// TIA Portal project "Hệ thống bơm cấp nước" (V16)

(* hardware
DEVICE "PC-System_1"  SIMATIC PC station
   slot 0: "SIMATIC PC station"  Rail  SIMATIC PC-Station  V1.0
      slot 125: "Stationmanager"  Station_Manager  V6.0.4
   slot 1: "HMI_RT_1"  WinCC RT Advanced  6AV2 104-0xxxx-xxxx  16.0.0.0
      slot 33792: "Computer interface"  Host interface
   slot 2: "IE general_1"  IE General  IE_CP  V8.2.0
DEVICE "S7-1200 station_1"  S7-1200 Station
   slot 0: "Rack_0"  S7-1200 Rack  Rack  V1.0
   slot 1: "PLC_1"  CPU 1214C DC/DC/DC  6ES7 214-1AG40-0XB0  V4.4
DEVICE "PC-System_2"  SIMATIC PC station
   slot 0: "SIMATIC PC station"  Rail  SIMATIC PC-Station  V1.0
      slot 125: "Stationmanager"  Station_Manager  V6.0.4
   slot 2: "IE general_1"  IE General  IE_CP  V8.2.0
*)

// ===== PLC "PLC_1"  CPU 1214C DC/DC/DC =====

VAR_GLOBAL   // PLC tag table "Default tag table"
   "START_VALVE_1" AT %M3.0 : Bool;
   "STOP_VALVE_1" AT %M3.1 : Bool;
   "START_VALVE_2" AT %M3.2 : Bool;
   "STOP_VALVE_2" AT %M3.3 : Bool;
   "START_PUMP_1" AT %M3.4 : Bool;
   "STOP_PUMP_1" AT %M3.5 : Bool;
   "START_PUMP_2" AT %M3.6 : Bool;
   "STOP_PUMP_2" AT %M3.7 : Bool;
   "START_PUMP_SUPPLY" AT %M4.0 : Bool;
   "STOP_PUMP_SUPPLY" AT %M4.1 : Bool;
   "VALVE_1" AT %Q0.0 : Bool;
   "VALVE_2" AT %Q0.1 : Bool;
   "PUMP_1" AT %Q0.2 : Bool;
   "PUMP_2" AT %Q0.3 : Bool;
   "PUMP_SUPPLY" AT %Q0.4 : Bool;
   "VALUE" AT %M4.2 : Bool;
   "SENSOR_1" AT %M4.3 : Bool;
   "SENSOR_2" AT %M4.4 : Bool;
   "SENSOR_3" AT %M4.5 : Bool;
   "TIME_RUN_PUMP 1" AT %MD10 : Time;
   "NO_WATER_PUMP_1" AT %M4.6 : Bool;
   "NO_WATER_PUMP_2" AT %M4.7 : Bool;
   "TIME_RUN_PUMP 2" AT %MD14 : Time;
   "System_Byte" AT %MB1 : Byte;
   "FirstScan" AT %M1.0 : Bool;
   "DiagStatusUpdate" AT %M1.1 : Bool;
   "AlwaysTRUE" AT %M1.2 : Bool;
   "AlwaysFALSE" AT %M1.3 : Bool;
   "Clock_Byte" AT %MB0 : Byte;
   "Clock_10Hz" AT %M0.0 : Bool;
   "Clock_5Hz" AT %M0.1 : Bool;
   "Clock_2.5Hz" AT %M0.2 : Bool;
   "Clock_2Hz" AT %M0.3 : Bool;
   "Clock_1.25Hz" AT %M0.4 : Bool;
   "Clock_1Hz" AT %M0.5 : Bool;
   "Clock_0.625Hz" AT %M0.6 : Bool;
   "Clock_0.5Hz" AT %M0.7 : Bool;
   "FULL_TANK_TOP" AT %M5.0 : Bool;
   "LEVEL_TANK_TOP" AT %MW18 : UInt;
   "EMPTY_TANK_TOP" AT %M5.1 : Bool;
   "FULL_TANK_BOT" AT %M5.2 : Bool;
   "USER" AT %MW22 : Word;
   "LEVEL_TANK_BOT" AT %MW20 : UInt;
   "EMPTY_TANK_BOT" AT %M5.3 : Bool;
END_VAR

// folder: System blocks/Program resources

DATA_BLOCK "IEC_Timer_0_DB"   // DB1
{ S7_Optimized_Access := 'TRUE' }
AUTHOR : Simatic
FAMILY : IEC
NAME : IEC_TMR
VERSION : 1.0
// stored: InstanceOfName IEC_TIMER
"IEC_TIMER"
BEGIN
END_DATA_BLOCK

DATA_BLOCK "IEC_Timer_0_DB_1"   // DB2
{ S7_Optimized_Access := 'TRUE' }
AUTHOR : Simatic
FAMILY : IEC
NAME : IEC_TMR
VERSION : 1.0
// stored: InstanceOfName IEC_TIMER
"IEC_TIMER"
BEGIN
END_DATA_BLOCK

DATA_BLOCK "IEC_Counter_0_DB"   // DB3
{ S7_Optimized_Access := 'TRUE' }
AUTHOR : Simatic
FAMILY : IEC
NAME : UCNTR
VERSION : 1.2
// stored: InstanceOfName IEC_UCOUNTER
"IEC_UCOUNTER"
BEGIN
END_DATA_BLOCK

DATA_BLOCK "IEC_Counter_0_DB_1"   // DB4
{ S7_Optimized_Access := 'TRUE' }
AUTHOR : Simatic
FAMILY : IEC
NAME : UCNTR
VERSION : 1.2
// stored: InstanceOfName IEC_UCOUNTER
"IEC_UCOUNTER"
BEGIN
END_DATA_BLOCK

// folder: (top level)

ORGANIZATION_BLOCK "Main"   // OB1, LAD, ProgramCycle
TITLE = Hệ thống cung cấp nước
{ S7_Optimized_Access := 'TRUE' }
VERSION : 0.1
   VAR_INPUT
      Initial_Call : Bool;   // Initial call of this OB
      Remanence : Bool;   // =True, if remanent data are available
   END_VAR
   VAR_TEMP
      EMPTY_TANK_BOT : Bool;
      LEVEL_TANK_BOT : Int;
   END_VAR
BEGIN

REGION Network 1: Control valve 1
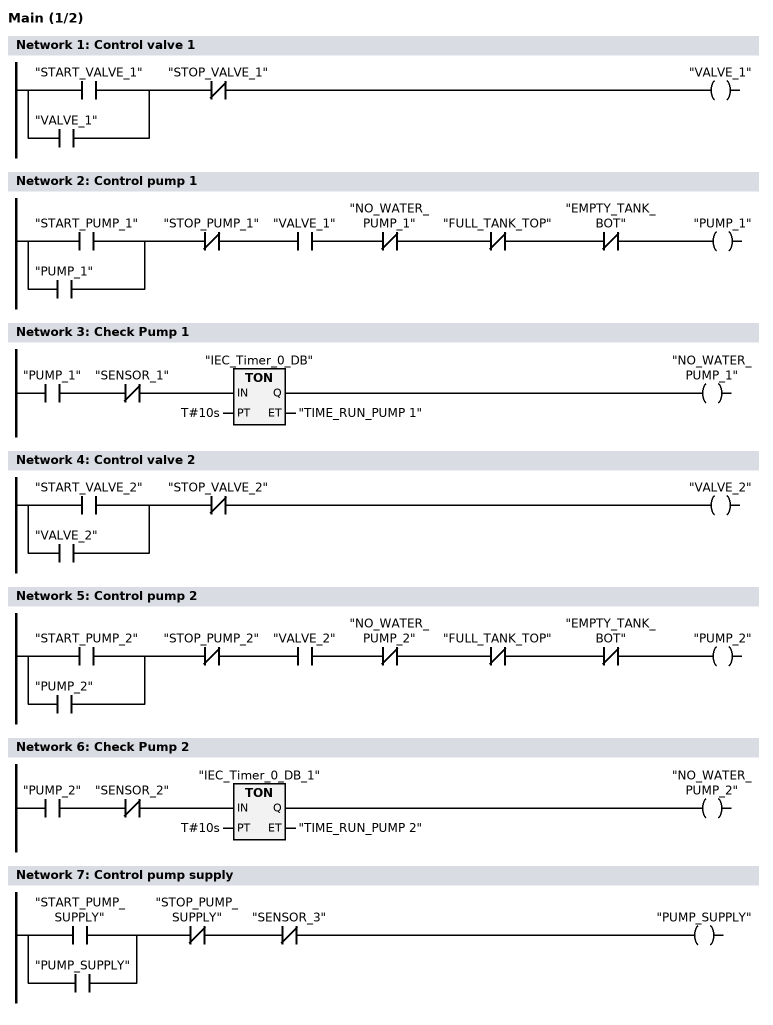
   RUNG wire#powerrail
      Contact( "START_VALVE_1" )
      wire#w1
      I_Contact( "STOP_VALVE_1" )
      Coil( "VALVE_1" )
   END_RUNG
   RUNG wire#powerrail
      Contact( "VALVE_1" )
   END_RUNG wire#w1
   // the same network as SCL:
   "VALVE_1" := ("START_VALVE_1" OR "VALVE_1") AND NOT "STOP_VALVE_1";
END_REGION

REGION Network 2: Control pump 1
   RUNG wire#powerrail
      Contact( "START_PUMP_1" )
      wire#w1
      I_Contact( "STOP_PUMP_1" )
      Contact( "VALVE_1" )
      I_Contact( "NO_WATER_PUMP_1" )
      I_Contact( "FULL_TANK_TOP" )
      I_Contact( "EMPTY_TANK_BOT" )
      Coil( "PUMP_1" )
   END_RUNG
   RUNG wire#powerrail
      Contact( "PUMP_1" )
   END_RUNG wire#w1
   // the same network as SCL:
   "PUMP_1" := ("START_PUMP_1" OR "PUMP_1") AND NOT "STOP_PUMP_1" AND "VALVE_1" AND NOT "NO_WATER_PUMP_1" AND NOT "FULL_TANK_TOP" AND NOT "EMPTY_TANK_BOT";
END_REGION

REGION Network 3: Check Pump 1
   "IEC_Timer_0_DB".TON(IN := "PUMP_1" AND NOT "SENSOR_1", PT := T#10s, ET => "TIME_RUN_PUMP 1");
   "NO_WATER_PUMP_1" := "IEC_Timer_0_DB".Q;
END_REGION

REGION Network 4: Control valve 2
   RUNG wire#powerrail
      Contact( "START_VALVE_2" )
      wire#w1
      I_Contact( "STOP_VALVE_2" )
      Coil( "VALVE_2" )
   END_RUNG
   RUNG wire#powerrail
      Contact( "VALVE_2" )
   END_RUNG wire#w1
   // the same network as SCL:
   "VALVE_2" := ("START_VALVE_2" OR "VALVE_2") AND NOT "STOP_VALVE_2";
END_REGION

REGION Network 5: Control pump 2
   RUNG wire#powerrail
      Contact( "START_PUMP_2" )
      wire#w1
      I_Contact( "STOP_PUMP_2" )
      Contact( "VALVE_2" )
      I_Contact( "NO_WATER_PUMP_2" )
      I_Contact( "FULL_TANK_TOP" )
      I_Contact( "EMPTY_TANK_BOT" )
      Coil( "PUMP_2" )
   END_RUNG
   RUNG wire#powerrail
      Contact( "PUMP_2" )
   END_RUNG wire#w1
   // the same network as SCL:
   "PUMP_2" := ("START_PUMP_2" OR "PUMP_2") AND NOT "STOP_PUMP_2" AND "VALVE_2" AND NOT "NO_WATER_PUMP_2" AND NOT "FULL_TANK_TOP" AND NOT "EMPTY_TANK_BOT";
END_REGION

REGION Network 6: Check Pump 2
   "IEC_Timer_0_DB_1".TON(IN := "PUMP_2" AND NOT "SENSOR_2", PT := T#10s, ET => "TIME_RUN_PUMP 2");
   "NO_WATER_PUMP_2" := "IEC_Timer_0_DB_1".Q;
END_REGION

REGION Network 7: Control pump supply
   RUNG wire#powerrail
      Contact( "START_PUMP_SUPPLY" )
      wire#w1
      I_Contact( "STOP_PUMP_SUPPLY" )
      I_Contact( "SENSOR_3" )
      Coil( "PUMP_SUPPLY" )
   END_RUNG
   RUNG wire#powerrail
      Contact( "PUMP_SUPPLY" )
   END_RUNG wire#w1
   // the same network as SCL:
   "PUMP_SUPPLY" := ("START_PUMP_SUPPLY" OR "PUMP_SUPPLY") AND NOT "STOP_PUMP_SUPPLY" AND NOT "SENSOR_3";
END_REGION

REGION Network 8: Simulation tank top
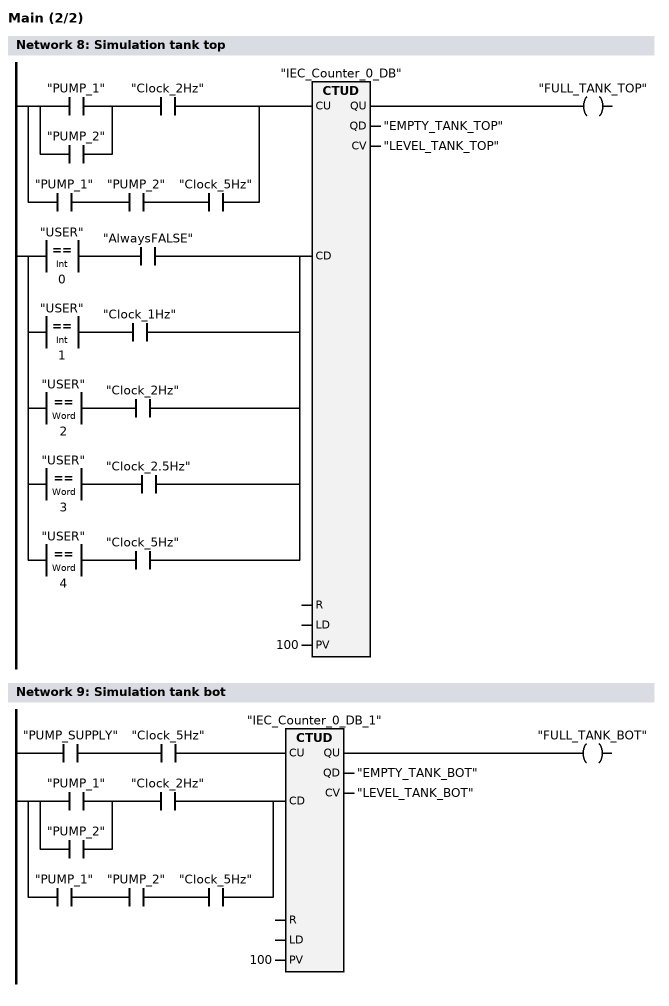
   "IEC_Counter_0_DB".CTUD(CU := (("PUMP_1" OR "PUMP_2") AND "Clock_2Hz") OR ("PUMP_1" AND "PUMP_2" AND "Clock_5Hz"),
                           CD := (("USER" = 0) AND "AlwaysFALSE") OR (("USER" = 1) AND "Clock_1Hz") OR (("USER" = 2) AND "Clock_2Hz") OR (("USER" = 3) AND "Clock_2.5Hz") OR (("USER" = 4) AND "Clock_5Hz"),
                           PV := 100,
                           QD => "EMPTY_TANK_TOP",
                           CV => "LEVEL_TANK_TOP");
   "FULL_TANK_TOP" := "IEC_Counter_0_DB".QU;
END_REGION

REGION Network 9: Simulation tank bot
   "IEC_Counter_0_DB_1".CTUD(CU := "PUMP_SUPPLY" AND "Clock_5Hz",
                           CD := (("PUMP_1" OR "PUMP_2") AND "Clock_2Hz") OR ("PUMP_1" AND "PUMP_2" AND "Clock_5Hz"),
                           PV := 100,
                           QD => "EMPTY_TANK_BOT",
                           CV => "LEVEL_TANK_BOT");
   "FULL_TANK_BOT" := "IEC_Counter_0_DB_1".QU;
END_REGION
END_ORGANIZATION_BLOCK

(* ===== HMI "HMI_RT_1" =====
system functions are stored by id; their names below are inferred from use
connection "HMI_Connection_1": ETHERNET, S7_1200_OMS

HMI tags "Default tag table"
   "START_VALVE_1" : Bool = PLC START_VALVE_1 AT %M3.0, 1 s
   "STOP_VALVE_1" : Bool = PLC STOP_VALVE_1 AT %M3.1, 1 s
   "START_VALVE_2" : Bool = PLC START_VALVE_2 AT %M3.2, 1 s
   "STOP_VALVE_2" : Bool = PLC STOP_VALVE_2 AT %M3.3, 1 s
   "START_PUMP_1" : Bool = PLC START_PUMP_1 AT %M3.4, 1 s
   "STOP_PUMP_1" : Bool = PLC STOP_PUMP_1 AT %M3.5, 1 s
   "START_PUMP_2" : Bool = PLC START_PUMP_2 AT %M3.6, 1 s
   "STOP_PUMP_2" : Bool = PLC STOP_PUMP_2 AT %M3.7, 1 s
   "START_PUMP_SUPPLY" : Bool = PLC START_PUMP_SUPPLY AT %M4.0, 1 s
   "STOP_PUMP_SUPPLY" : Bool = PLC STOP_PUMP_SUPPLY AT %M4.1, 1 s
   "VALVE_1" : Bool = PLC VALVE_1 AT %Q0.0, 1 s
   "VALVE_2" : Bool = PLC VALVE_2 AT %Q0.1, 1 s
   "PUMP_1" : Bool = PLC PUMP_1 AT %Q0.2, 1 s
   "PUMP_2" : Bool = PLC PUMP_2 AT %Q0.3, 1 s
   "PUMP_SUPPLY" : Bool = PLC PUMP_SUPPLY AT %Q0.4, 1 s
   "VALUE" : Bool = PLC VALUE AT %M4.2, 1 s
   "SENSOR_1" : Bool = PLC SENSOR_1 AT %M4.3, 1 s
   "SENSOR_2" : Bool = PLC SENSOR_2 AT %M4.4, 1 s
   "SENSOR_3" : Bool = PLC SENSOR_3 AT %M4.5, 1 s
   "TIME_RUN_PUMP 1" : Time = PLC "TIME_RUN_PUMP 1" AT %MD10, 1 s
   "TIME_RUN_PUMP 2" : Time = PLC "TIME_RUN_PUMP 2" AT %MD14, 1 s
   "LEVEL_TANK" : UInt = PLC LEVEL_TANK_TOP AT %MW18, 1 s
   "LEVEL_TANK_BOT" : UInt = PLC LEVEL_TANK_BOT AT %MW20, 1 s
   "USER" : Word = PLC USER AT %MW22, 1 s

text list "Text_list_1": 0 '0%'; 1 '10%'; 2 '20%'; 3 '30%'; 4 '40%'

screen "Screen_1" 1080x1920
   SymbolLibrary "Symbol library_4" at 372,310 size 62x53
      Appearance <- "PUMP_2"
   SymbolLibrary "Symbol library_8" at 414,175 size 16x152
   SymbolLibrary "Symbol library_1" at 601,200 size 303x280
   SymbolLibrary "Symbol library_2" at 612,49 size 120x171
   Bar "Bar_1" at 204,373 size 343x158; MinimumValue 0; MaximumValue 100
      ProcessValue <- "LEVEL_TANK_BOT"
   Bar "Bar_2" at 633,51 size 80x138; MinimumValue 0; MaximumValue 100
      ProcessValue <- "LEVEL_TANK"
   SymbolLibrary "Symbol library_3" at 442,151 size 174x15
   SymbolLibrary "Symbol library_5" at 483,141 size 27x27
   SymbolLibrary "Symbol library_6" at 414,151 size 30x29
   SymbolLibrary "Symbol library_7" at 413,177 size 46x38
      Appearance <- "VALVE_2"
   SymbolLibrary "Symbol library_9" at 430,333 size 47x15
   SymbolLibrary "Symbol library_10" at 474,333 size 35x29
   SymbolLibrary "Symbol library_11" at 491,360 size 18x17
   SymbolLibrary "Symbol library_12" at 145,311 size 62x53
      Appearance <- "PUMP_1"
   SymbolLibrary "Symbol library_13" at 203,334 size 47x15
   SymbolLibrary "Symbol library_14" at 247,334 size 35x29
   SymbolLibrary "Symbol library_15" at 264,361 size 18x15
   SymbolLibrary "Symbol library_16" at 188,119 size 16x216
   SymbolLibrary "Symbol library_17" at 188,93 size 31x30
   SymbolLibrary "Symbol library_18" at 187,185 size 46x38
      Appearance <- "VALVE_1"
   SymbolLibrary "Symbol library_19" at 214,93 size 400x16
   SymbolLibrary "Symbol library_20" at 259,83 size 27x29
   SymbolLibrary "Symbol library_21" at 237,41 size 21x52
      Appearance <- "SENSOR_1"
      on Click: InvertBit("SENSOR_1")
   SymbolLibrary "Symbol library_23" at 145,377 size 59x26
      Appearance <- "SENSOR_3"
      on Click: InvertBit("SENSOR_3")
   SymbolLibrary "Symbol library_24" at 134,456 size 72x66
      Appearance <- "PUMP_SUPPLY"
   TextField "Text field_1" at 63,378 size 71x22; Text 'Sensor 3'
   TextField "Text field_2" at 70,325 size 64x22; Text 'Pump 1'
   TextField "Text field_3" at 332,303 size 52x20; Text 'Pump 2'
   TextField "Text field_4" at 119,199 size 61x22; Text 'Valve 1'
   TextField "Text field_5" at 349,185 size 61x22; Text 'Valve 2'
   TextField "Text field_6" at 163,46 size 71x22; Text 'Sensor 1'
   TextField "Text field_7" at 354,123 size 71x22; Text 'Sensor 2'
   TextField "Text field_8" at 105,521 size 92x22; Text 'Pump Suply'
   Button "Button_1" at 38,286 size 53x32; TextOff 'Start'
      on Press: SetBit("START_PUMP_1")
      on Release: ResetBit("START_PUMP_1")
   Button "Button_2" at 92,286 size 53x32; TextOff 'Stop'
      on Release: ResetBit("STOP_PUMP_1")
      on Press: SetBit("STOP_PUMP_1")
   Button "Button_3" at 300,271 size 53x32; TextOff 'Start'
      on Release: ResetBit("START_PUMP_2")
      on Press: SetBit("START_PUMP_2")
   Button "Button_4" at 354,271 size 53x32; TextOff 'Stop'
      on Release: ResetBit("STOP_PUMP_2")
      on Press: SetBit("STOP_PUMP_2")
   Button "Button_5" at 95,539 size 53x32; TextOff 'Start'
      on Release: ResetBit("START_PUMP_SUPPLY")
      on Press: SetBit("START_PUMP_SUPPLY")
   Button "Button_6" at 149,539 size 53x32; TextOff 'Stop'
      on Release: ResetBit("STOP_PUMP_SUPPLY")
      on Press: SetBit("STOP_PUMP_SUPPLY")
   Button "Button_7" at 78,157 size 53x32; TextOff 'Start'
      on Release: ResetBit("START_VALVE_1")
      on Press: SetBit("START_VALVE_1")
   Button "Button_8" at 132,157 size 53x32; TextOff 'Stop'
      on Release: ResetBit("STOP_VALVE_1")
      on Press: SetBit("STOP_VALVE_1")
   Button "Button_9" at 461,177 size 53x32; TextOff 'Start'
      on Release: ResetBit("START_VALVE_2")
      on Press: SetBit("START_VALVE_2")
   Button "Button_10" at 515,177 size 53x32; TextOff 'Stop'
      on Release: ResetBit("STOP_VALVE_2")
      on Press: SetBit("STOP_VALVE_2")
   IOField "I/O field_1" at 257,41 size 96x32; FormatPattern 999999
      ProcessValue <- "TIME_RUN_PUMP 1"
   SymbolicIOField "Symbolic I/O field_1" at 732,93 size 96x32; TextOff '0'; TextOn '1'; TextList "Text_list_1"
      ProcessValue <- "USER"
   TextField "Text field_9" at 430,16 size 163x20; Text 'Hệ thống bơm nước'
   IOField "I/O field_2" at 461,109 size 96x32; FormatPattern s9999999999
      ProcessValue <- "TIME_RUN_PUMP 2"
   SymbolLibrary "Symbol library_22" at 433,99 size 22x52
      on Click: InvertBit("SENSOR_2")
      Appearance <- "SENSOR_2"
*)